TYPE ST_OutfeedConveyorMachPar :
STRUCT
	VelocityManual						: LREAL;
	VelocityAuto						: LREAL;
	
END_STRUCT
END_TYPE

(* stored: Version 1.1.0.1, ProductVersion 3.1.4020.12
   DUT ST_OutfeedConveyorMachPar: Id {83d35d86-a911-4b17-9794-36fec88beb43} *)
